Omron CX-Programmer project Carrinho_areia (CX-Programmer 9.81)

# PLC NewPLC2: CJ1M CPU11
I/O table (CPU CJ1M-CPU11): rack 0 slot 0 CJ1W-ID211; rack 0 slot 1 CJ1W-OD211

## Program NewProgram1 (cyclic task 0)
Local symbols
botao_de_emergência 0.02 BOOL  ; botao de emergencia
botão_start 0.00 BOOL  ; botao start
botão_stop 0.01 BOOL  ; botao stop
etapa_1 2.00 BOOL  ; etapa1 grafcet
etapa_2 2.01 BOOL  ; etapa2 grafcet
etapa_3 2.02 BOOL  ; etapa3 grafcet
etapa_4 2.03 BOOL  ; etapa4 grafcet
etapa_5 2.04 BOOL  ; etapa5 grafcet
etapa_6 2.05 BOOL  ; etapa6 grafcet
flag_t1 T0001 BOOL  ; flag do temporizador 1
flag_t2 T0002 BOOL  ; flag do temporizador 2
km1_d 1.00 BOOL  ; motor direita
km2_e 1.01 BOOL  ; motor esquerda
km3_stop 1.03 BOOL  ; motor para
s_A 0.04 BOOL  ; sensor fdc esquerda
s_B 0.05 BOOL  ; sensor fdc direita
sensor_balança 0.03 BOOL  ; sensor balança
t_02 2 NUMBER  ; temporizador 2
t_1 1 NUMBER  ; temporizador 1
tempo_t1 #10 NUMBER  ; tempo do temporizador 1
tempo_t2 #40 NUMBER  ; tempo do temporizador 2
valvula_abre 1.02 BOOL  ; valvula
valvula_fecha 1.04 BOOL  ; valvula fecha

### Section OUT

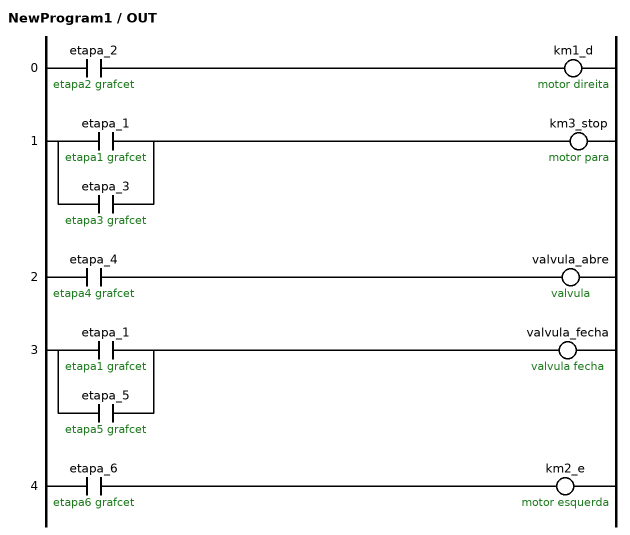
; rung 0
LD etapa_2  ; etapa2 grafcet
OUT km1_d  ; motor direita
; rung 1
LD etapa_1  ; etapa1 grafcet
OR etapa_3  ; etapa3 grafcet
OUT km3_stop  ; motor para
; rung 2
LD etapa_4  ; etapa4 grafcet
OUT valvula_abre  ; valvula
; rung 3
LD etapa_1  ; etapa1 grafcet
OR etapa_5  ; etapa5 grafcet
OUT valvula_fecha  ; valvula fecha
; rung 4
LD etapa_6  ; etapa6 grafcet
OUT km2_e  ; motor esquerda

### Section MAIN

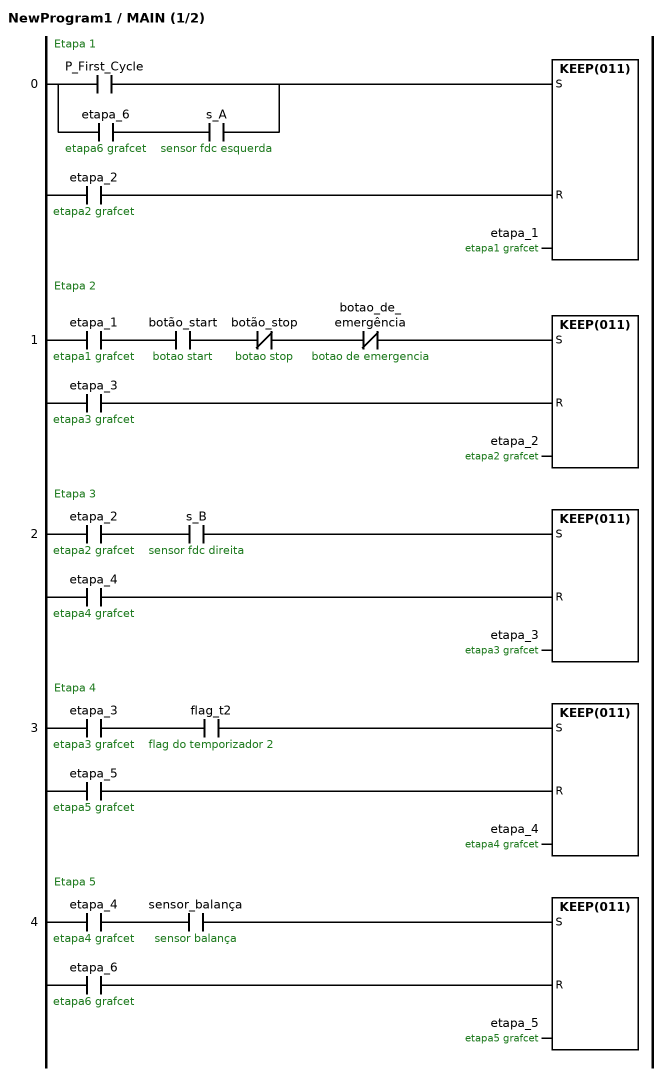
; rung 0: Etapa 1
LD P_First_Cycle
LD etapa_6  ; etapa6 grafcet
AND s_A  ; sensor fdc esquerda
ORLD
LD etapa_2  ; etapa2 grafcet
KEEP(011) etapa_1  ; etapa1 grafcet
; rung 1: Etapa 2
LD etapa_1  ; etapa1 grafcet
AND botão_start  ; botao start
ANDNOT botão_stop  ; botao stop
ANDNOT botao_de_emergência  ; botao de emergencia
LD etapa_3  ; etapa3 grafcet
KEEP(011) etapa_2  ; etapa2 grafcet
; rung 2: Etapa 3
LD etapa_2  ; etapa2 grafcet
AND s_B  ; sensor fdc direita
LD etapa_4  ; etapa4 grafcet
KEEP(011) etapa_3  ; etapa3 grafcet
; rung 3: Etapa 4
LD etapa_3  ; etapa3 grafcet
AND flag_t2  ; flag do temporizador 2
LD etapa_5  ; etapa5 grafcet
KEEP(011) etapa_4  ; etapa4 grafcet
; rung 4: Etapa 5
LD etapa_4  ; etapa4 grafcet
AND sensor_balança  ; sensor balança
LD etapa_6  ; etapa6 grafcet
KEEP(011) etapa_5  ; etapa5 grafcet

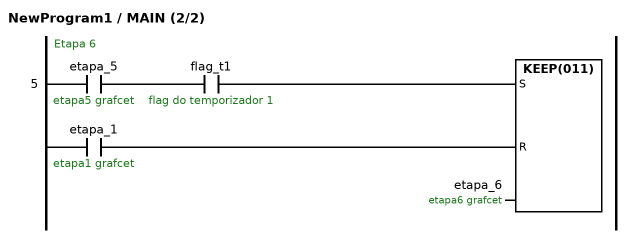
; rung 5: Etapa 6
LD etapa_5  ; etapa5 grafcet
AND flag_t1  ; flag do temporizador 1
LD etapa_1  ; etapa1 grafcet
KEEP(011) etapa_6  ; etapa6 grafcet

### Section Timers

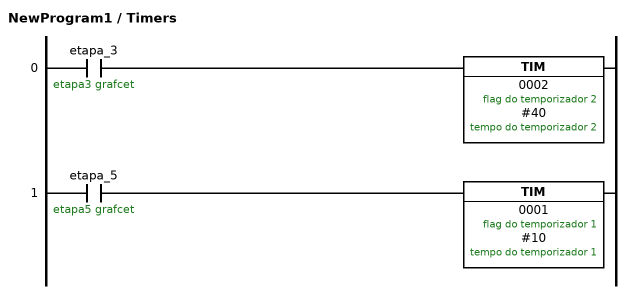
; rung 0
LD etapa_3  ; etapa3 grafcet
TIM 0002 #40  ; tempo do temporizador 2, flag do temporizador 2
; rung 1
LD etapa_5  ; etapa5 grafcet
TIM 0001 #10  ; tempo do temporizador 1, flag do temporizador 1

### Section END
; rung 0
END(001)